{attribute 'qualified_only'}
VAR_GLOBAL
END_VAR

(* stored: Version 1.1.0.1, ProductVersion 3.1.4024.16
   GVL vb: Id {26e8e9e1-7cb9-4761-92d4-188c5c0ae794} *)
